ELSIF m_scopeArmIndex = m_matchedMasterArmIdx.right1ArmIdx OR m_scopeArmIndex = m_matchedMasterArmIdx.right2ArmIdx THEN
	// left arm
	// switch tele-controlled arm index when arm switch is triggerd
	IF m_armSwitch THEN
		IF m_teleSlaveArmIdx[1]=m_matchedMasterArmIdx.left1ArmIdx AND i_masterInputDataPool.m_slaveStatus.m_armState[m_matchedMasterArmIdx.left2ArmIdx]=SlaveArmState_InstruReady THEN
			nextTeleSlaveArmIdx[1] := m_matchedMasterArmIdx.left2ArmIdx;
		ELSIF 
			m_teleSlaveArmIdx[1]=m_matchedMasterArmIdx.left2ArmIdx AND i_masterInputDataPool.m_slaveStatus.m_armState[m_matchedMasterArmIdx.left1ArmIdx]=SlaveArmState_InstruReady THEN
			nextTeleSlaveArmIdx[1] := m_matchedMasterArmIdx.left1ArmIdx;
		ELSE
			IF  i_masterInputDataPool.m_slaveStatus.m_armState[m_matchedMasterArmIdx.left1ArmIdx]=SlaveArmState_InstruReady THEN
				nextTeleSlaveArmIdx[1] := m_matchedMasterArmIdx.left1ArmIdx;
			ELSIF i_masterInputDataPool.m_slaveStatus.m_armState[m_matchedMasterArmIdx.left2ArmIdx]=SlaveArmState_InstruReady THEN
				nextTeleSlaveArmIdx[1] := m_matchedMasterArmIdx.left2ArmIdx;
			ELSE
				nextTeleSlaveArmIdx[1] := m_matchedMasterArmIdx.left1ArmIdx;
			END_IF
		END_IF
	END_IF

	// right arm
	IF m_scopeArmIndex = m_matchedMasterArmIdx.right1ArmIdx THEN
		nextTeleSlaveArmIdx[2] := m_matchedMasterArmIdx.right2ArmIdx;
	ELSE
		nextTeleSlaveArmIdx[2] := m_matchedMasterArmIdx.right1ArmIdx;
	END_IF
END_IF

// check if arm-switch is triggerd
m_armSwitchFlag[1]:=m_teleSlaveArmIdx[1] <>  nextTeleSlaveArmIdx[1];
m_armSwitchFlag[2]:=m_teleSlaveArmIdx[2] <>  nextTeleSlaveArmIdx[2];

m_teleSlaveArmIdx:= nextTeleSlaveArmIdx;
END_METHOD

METHOD PROTECTED controllerTransit : BOOL
VAR_INPUT
END_VAR
VAR
	i :INT;
END_VAR
FOR i:=1 TO g_mArmNum DO 
	IF m_nextMasterArmState[i]<> m_masterArmState[i] THEN
		// reset current controller
		m_armCtrl[i].reset();
		
		// transit to new controller
		m_lastMasterArmState[i]:=m_masterArmState[i];
		m_masterArmState[i]:=m_nextMasterArmState[i];
		m_armCtrl[i]:=m_armCtrlFactory[i,m_masterArmState[i]];
		
		// init next controller
		m_armCtrl[i].Init(m_masterArms[i],m_armCtrlCmds[i]);
		
		// init scope controller
		IF m_masterArmState[i] = MasterArmState_Endoscope  THEN
			m_scopeCtrl.init(m_shoulderPoseInMonitor, m_masterArms, m_armCtrlCmds);
		END_IF
		
		m_masterArms[i].updateCmds(m_armCtrlCmds[i]);
	END_IF
END_FOR
END_METHOD

METHOD PUBLIC getStatus : BOOL
VAR_IN_OUT
	// master robot information, including arm status and cartesian data
	r_masterStatus :ST_MasterStatus;
	
	// master robot joint data
	r_masterJointsData :ST_MasterJointData;
	
END_VAR

VAR
	i:INT;
END_VAR
r_masterStatus.m_motionScale := m_motionScale;
r_masterStatus.m_armState:=m_masterArmState;
r_masterStatus.m_teleSlaveArmIdx := m_teleSlaveArmIdx;
r_masterStatus.m_matchedMasterArmIdx := m_matchedMasterArmIdx;

FOR i:=1 TO g_mArmNum DO
	// current info
	r_masterStatus.m_gripAngle[i]:=m_masterArms[i].gripAngle;
	// cartesion
	r_masterStatus.m_curArmPose[i]:=m_masterArms[i].curCartPose;
	r_masterStatus.m_curArmTwist[i]:=m_masterArms[i].curCartTwist;
	// joint
	r_masterJointsData.m_curMotorPos[i]:=m_masterArms[i].curMotorPos;
	r_masterJointsData.m_curLinkPos[i]:=m_masterArms[i].curLinkPos;
	r_masterJointsData.m_curJntPos[i]:=m_masterArms[i].curJntPos;
	r_masterJointsData.m_curJntVel[i]:=m_masterArms[i].curJntVel;
	r_masterJointsData.m_curJntTrq[i]:=m_masterArms[i].curJntTrq;
	r_masterJointsData.m_rawJntCurrent[i]:=m_masterArms[i].rawJntCurrent;
	r_masterJointsData.m_filtJntCurrent[i]:=m_masterArms[i].filtJntCurrent;
	
	// command info
	// cartesion
	r_masterStatus.m_cmdArmPose[i]:=m_masterArms[i].m_cmdCartPose;
	r_masterStatus.m_cmdArmTwist[i]:=m_masterArms[i].m_cmdCartTwist;
	// joint info
	r_masterJointsData.m_cmdJntPos[i]:=m_masterArms[i].m_cmdJntPos;
	r_masterJointsData.m_cmdJntVel[i]:=m_masterArms[i].m_cmdJntVel;
	r_masterJointsData.m_cmdJntTrq[i]:=m_masterArms[i].m_cmdJntTrq;
	r_masterJointsData.m_cmdJntCurrent[i]:=m_masterArms[i].cmdJntCurrent;
	//data to safety check
	r_masterStatus.m_gripHallSensor[i] := m_masterArms[i].m_gripHallSensorIO;
	r_masterStatus.m_slaveOnLine := m_slaveOnLine;
	r_masterStatus.m_IKSuccess[i] := m_armMatching[i].IKSuccess;
	r_masterStatus.m_timePeriod[i] := m_armMatching[i].timePeriod;
	//r_masterStatus.m_selfCheckStatus
END_FOR
END_METHOD

METHOD PUBLIC Init : BOOL
VAR_INPUT
END_VAR
VAR
	i:INT;
END_VAR
// init tele-controlled arm index
m_teleSlaveArmIdx[1]:=MatchedSlaveArmIdx_1;
m_teleSlaveArmIdx[2]:=MatchedSlaveArmIdx_3;

// shoulder pose in monitor
m_shoulderPoseInMonitor[1].m_pos[1]:=-g_shoulderDistance/2;
m_shoulderPoseInMonitor[2].m_pos[1]:=g_shoulderDistance/2;

FOR i:=1 TO g_mArmNum DO
	// arm init
	m_masterArms[i].Init(i);
	m_masterArmState[i]:=MasterArmState_Init;
	m_lastMasterArmState[i]:=MasterArmState_Init;
	m_nextMasterArmState[i]:=MasterArmState_Init;
	
	// command init
	m_armCtrlCmds[i].m_jntEnableFlag := g_zeroVec7i;
	m_armCtrlCmds[i].m_jntOPMode := g_allPosMode;
	m_armCtrlCmds[i].m_cmdCartPose := m_masterArms[i].curCartPose;
	m_armCtrlCmds[i].m_cmdCartTwist := g_zeroVec6d;
	m_armCtrlCmds[i].m_cmdJntPos := m_masterArms[i].curJntPos;
	m_armCtrlCmds[i].m_cmdJntVel := g_zeroVec7d;
	m_armCtrlCmds[i].m_cmdJntAcc := g_zeroVec7d;
	m_armCtrlCmds[i].m_cmdJntTrq := g_zeroVec7d;
	
	// generate controller factory
	m_armCtrlFactory[i,MasterArmState_Error] := m_armError[i];
	m_armCtrlFactory[i,MasterArmState_Init] := m_armInit[i];
	m_armCtrlFactory[i,MasterArmState_Home] := m_armHome[i];
	m_armCtrlFactory[i,MasterArmState_Standby] := m_armStandBy[i];
	m_armCtrlFactory[i,MasterArmState_Matching] := m_armMatching[i];
	m_armCtrlFactory[i,MasterArmState_Ready] := m_armReady[i];
	m_armCtrlFactory[i,MasterArmState_MasterSlave] := m_armMasterSlave[i];
	m_armCtrlFactory[i,MasterArmState_Clutch] := m_armClutch[i];
	m_armCtrlFactory[i,MasterArmState_Endoscope] := m_armEndoscope[i];
	m_armCtrlFactory[i,MasterArmState_Cart] := m_armCart[i];
	m_armCtrlFactory[i,MasterArmState_GravityCali] := m_armGravityCali[i];
	m_armCtrlFactory[i,MasterArmState_Test] := m_armTest[i];
	m_armCtrlFactory[i,MasterArmState_Disable] := m_armDisable[i];
	m_armCtrlFactory[i,MasterArmState_Performance] := m_armPerformance[i];

	// assign controller
	m_armCtrl[i]:=m_armCtrlFactory[i,m_masterArmState[i]];
	m_armCtrl[i].Init(m_masterArms[i],m_armCtrlCmds[i]);
	
	// init master-slave trigger
	m_MSCtrlTriggerCheck[i].init(g_armCtrlCycleTime, 2);
END_FOR
END_METHOD

METHOD PROTECTED MSCtrlTriggerCheck : BOOL
VAR_IN_OUT CONSTANT
		i_masterInputDataPool:ST_MasterInputDataPool;
END_VAR
VAR
	i:INT;
END_VAR
FOR i:=1 TO g_mArmNum DO
	IF MasterArmState_Ready = m_masterArmState[i] AND SlaveArmState_InstruReady = m_instruArmState[i] 
		AND SlaveArmState_ScopeReady = m_scopeArmState AND i_masterInputDataPool.m_cartStatus.m_surgonReady THEN
		m_MSCtrlTriggerFlag[i]:=m_MSCtrlTriggerCheck[i].run(m_masterArms[i].gripAngle);
	END_IF
	
	IF  MatchedSlaveArmIdx_NULL =  m_teleSlaveArmIdx[i] OR   NOT(i_masterInputDataPool.m_cartStatus.m_surgonReady) 
		OR 	NOT(i_masterInputDataPool.m_slaveStatus.m_instruStauts[m_teleSlaveArmIdx[i]].m_ready) 
		OR m_masterArmState[i] = MasterArmState_Error OR i_masterInputDataPool.m_cartStatus.m_consoleInAdjust
		OR  SlaveArmState_Error = m_instruArmState[i] OR SlaveArmState_Disable = m_instruArmState[i]  THEN
		m_MSCtrlTriggerFlag[i]:=FALSE;
		m_MSCtrlTriggerCheck[i].reset();
	END_IF  
END_FOR
END_METHOD

METHOD PUBLIC run : BOOL
VAR_IN_OUT CONSTANT
	i_masterInputDataPool:ST_MasterInputDataPool;
END_VAR
VAR
	i:INT;
END_VAR
m_motionScale := i_masterInputDataPool.m_UIData.m_motionScale;
m_monitorAngle := i_masterInputDataPool.m_cartStatus.m_monitorAngle;

// check slave connection
m_slaveOnLine := m_slaveOnLineCheck.check(i_masterInputDataPool.m_slaveStatus.m_slaveHeartBeat);

// update shoulder pose
updateShoulderPose();

// check tele-operated slave arms index
checkTeleSlaveArmIdx(i_masterInputDataPool);

// check if to trig ultrasonic knife ratotation clutch
USKnifeClutchCheck(i_masterInputDataPool);

// update arm status
FOR i:=1 TO g_mArmNum DO
	// update dynamic data
	m_masterArms[i].updateDyna(i_masterInputDataPool.m_masterDynaData);
								
	// update master arm kinematics
	m_masterArms[i].updateStatus();
END_FOR

// state machine transition
stateMachine(i_masterInputDataPool);

// controller transition
controllerTransit();

// run arm controller
FOR i:=1 TO g_mArmNum DO
	// null ptr check
	ASSERT(0 <> m_armCtrl[i]);
	
	// run controller
	m_armCtrl[i].run(m_teleSlaveArmIdx[i], m_shoulderPoseInMonitor[i], m_masterArms[i],
						i_masterInputDataPool.m_slaveStatus,m_armCtrlCmds[i]);
						
	// update commands to drivers
	m_masterArms[i].updateCmds(m_armCtrlCmds[i]);
END_FOR

// run scope controller
IF m_masterArmState[1] = MasterArmState_Endoscope AND m_masterArmState[2] = MasterArmState_Endoscope THEN
	m_scopeCtrl.run(m_teleSlaveArmIdx, m_shoulderPoseInMonitor, m_masterArms, i_masterInputDataPool.m_slaveStatus, m_armCtrlCmds);
	m_masterArms[1].updateCmds(m_armCtrlCmds[1]);
	m_masterArms[2].updateCmds(m_armCtrlCmds[2]);
END_IF
END_METHOD

PROPERTY shoulderPose : ARRAY[1..2] OF ST_Frame
GET
shoulderPose := m_shoulderPoseInMonitor;
END_GET
END_PROPERTY

// state machine check and transit 
METHOD PROTECTED stateMachine : BOOL
VAR_IN_OUT CONSTANT
		i_masterInputDataPool:ST_MasterInputDataPool;
END_VAR
VAR
	i:INT;
	enableClutch :BOOL;
END_VAR
// get instrument arm state
FOR i:=1 TO g_mArmNum DO
	IF MatchedSlaveArmIdx_NULL =  m_teleSlaveArmIdx[i] THEN
		m_instruArmState[i] := SlaveArmState_Error;
	ELSE
		m_instruArmState[i] := i_masterInputDataPool.m_slaveStatus.m_armState[m_teleSlaveArmIdx[i]];
	END_IF
END_FOR

// get endoscope arm state
m_scopeArmState := SlaveArmState_Error;
m_scopeArmIndex := MatchedSlaveArmIdx_null;
FOR i:=1 TO g_sArmNum DO 
	IF InstruType_endoscope =  i_masterInputDataPool.m_slaveStatus.m_instruStauts[i].m_type THEN
		m_scopeArmState := i_masterInputDataPool.m_slaveStatus.m_armState[i];
		m_scopeArmIndex := i;
		EXIT;
	END_IF
END_FOR

// check if master-slave grip angle match
MSCtrlTriggerCheck(i_masterInputDataPool);

// State machine transit 
FOR i:=1 TO g_mArmNum DO
	
	// flag if enable clutch
	enableClutch :=  i_masterInputDataPool.m_cartStatus.m_clutchSwitch OR (m_masterArms[i].handClutchSwitch AND i_masterInputDataPool.m_UIData.m_enableHandClutch);
	
	CASE m_masterArmState[i] OF
		// error
		MasterArmState_Error:
			// to standby
			IF FALSE = i_masterInputDataPool.m_safetyData.m_masterErrFlag[i] THEN
				IF m_armSelfCheckFinshedFlag[i] THEN
					m_nextMasterArmState[i] := MasterArmState_Standby;
				ELSE
					m_nextMasterArmState[i]:=MasterArmState_Home;
				END_IF
			END_IF
			
		// init
		MasterArmState_Init:
			// to home
			IF m_armCtrl[i].isFinished THEN
				// NOTICE: multiple cycles joints back to center during initialization
				// 			need to reset joints encoder data again
				m_masterArms[i].initJntPos();
				m_armSelfCheckFinshedFlag[i] := FALSE;
				m_nextMasterArmState[i]:=MasterArmState_Home;
			END_IF

		//home
		MasterArmState_Home:
			IF m_armCtrl[i].isFinished  THEN
				m_armSelfCheckFinshedFlag[i] := TRUE;
				m_nextMasterArmState[i]:=MasterArmState_Standby;
			END_IF
		
		//standby
		MasterArmState_Standby:
			// to matching
			IF SlaveArmState_InstruReady = m_instruArmState[i] AND SlaveArmState_ScopeReady = m_scopeArmState 
					AND i_masterInputDataPool.m_slaveStatus.m_asepticDeployCompleteFlag AND m_slaveOnLine THEN
				m_nextMasterArmState[i]:=MasterArmState_Matching;
			// to clutch
			ELSIF enableClutch THEN
				m_nextMasterArmState[i] := MasterArmState_Clutch; 
			// to cart
			ELSIF i_masterInputDataPool.m_cartStatus.m_monitorInAdjust THEN
				m_nextMasterArmState[i] := MasterArmState_Cart;
			END_IF
		
		//matching
		MasterArmState_Matching:
			// to ready
			IF m_armCtrl[i].isFinished THEN
				m_nextMasterArmState[i]:=MasterArmState_Ready;
			// to clutch
			ELSIF enableClutch THEN
				m_nextMasterArmState[i] := MasterArmState_Clutch; 
			// to standby
			ELSIF SlaveArmState_InstruReady <> m_instruArmState[i] OR SlaveArmState_ScopeReady <> m_scopeArmState
						OR m_armSwitchFlag[i] THEN
				m_nextMasterArmState[i]:=MasterArmState_Standby;
			// to cart
			ELSIF i_masterInputDataPool.m_cartStatus.m_monitorInAdjust THEN
				m_nextMasterArmState[i] := MasterArmState_Cart;
			END_IF
		
		//ready
		MasterArmState_Ready:
			// to standby
			IF SlaveArmState_InstruReady <> m_instruArmState[i] OR SlaveArmState_ScopeReady <> m_scopeArmState
					OR m_armSwitchFlag[i] THEN
				m_nextMasterArmState[i]:=MasterArmState_Standby;
			// to clutch
			ELSIF enableClutch THEN
				m_nextMasterArmState[i] := MasterArmState_Clutch; 
			// to cart
			ELSIF i_masterInputDataPool.m_cartStatus.m_monitorInAdjust THEN
				m_nextMasterArmState[i] := MasterArmState_Cart;
			// to master-slave
			ELSIF SlaveArmState_InstruReady = m_instruArmState[i] AND SlaveArmState_ScopeReady = m_scopeArmState 
					AND i_masterInputDataPool.m_cartStatus.m_surgonReady AND m_MSCtrlTriggerFlag[i] AND NOT(i_masterInputDataPool.m_cartStatus.m_consoleInAdjust) THEN
				m_nextMasterArmState[i] := MasterArmState_MasterSlave;
			ELSIF NOT i_masterInputDataPool.m_slaveStatus.m_asepticDeployCompleteFlag THEN
				m_nextMasterArmState[i]:=MasterArmState_Standby;
			END_IF
		
		//MasterSlave
		MasterArmState_MasterSlave:
			// to standdy
			IF  (SlaveArmState_InstruReady <> m_instruArmState[i] AND SlaveArmState_MasterSlave <> m_instruArmState[i])
				OR SlaveArmState_ScopeReady <> m_scopeArmState OR NOT(i_masterInputDataPool.m_cartStatus.m_surgonReady)
				OR m_armSwitchFlag[i] THEN
				m_nextMasterArmState[i]:=MasterArmState_Standby;
			// to clutch
			ELSIF enableClutch THEN
				m_nextMasterArmState[i] := MasterArmState_Clutch; 
			//to standby
			ELSIF NOT m_slaveOnLine THEN
				m_nextMasterArmState[i] := MasterArmState_Standby;
			END_IF
			
		//Clutch
		MasterArmState_Clutch:
			// to standby
			IF NOT(enableClutch) THEN
				m_nextMasterArmState[i]:=MasterArmState_Standby;
			END_IF
		
		// Endoscope 
		MasterArmState_Endoscope:
			// to standby
			IF NOT(i_masterInputDataPool.m_cartStatus.m_surgonReady) OR NOT(i_masterInputDataPool.m_cartStatus.m_endoscopeSwitch) 
				OR (SlaveArmState_ScopeReady <> m_scopeArmState AND SlaveArmState_EndoScope <> m_scopeArmState) THEN
				m_nextMasterArmState[i] := MasterArmState_Standby;
			// to clutch
			ELSIF enableClutch THEN
				m_nextMasterArmState[i] := MasterArmState_Clutch; 
			// to cart
			ELSIF i_masterInputDataPool.m_cartStatus.m_consoleInAdjust THEN
				m_nextMasterArmState[i] := MasterArmState_Cart;
			//to standby
			ELSIF NOT m_slaveOnLine THEN
				m_nextMasterArmState[i] := MasterArmState_Standby;
			END_IF
			
		// Cart 
		MasterArmState_Cart:
			// to standby
			IF NOT( i_masterInputDataPool.m_cartStatus.m_consoleInAdjust) THEN
				m_nextMasterArmState[i] := MasterArmState_Standby;
			END_IF
		
		//Gravity Calibration
		MasterArmState_GravityCali:
			// to standby
			IF  m_armCtrl[i].isFinished THEN
				m_nextMasterArmState[i]:=MasterArmState_Standby;
			END_IF
	
		//arm test
		MasterArmState_Test:
			// to standby
			IF  m_armCtrl[i].isFinished THEN
				m_nextMasterArmState[i]:=MasterArmState_Standby;
			END_IF
			
		//arm Performance
		MasterArmState_Performance:
			// to standby
			IF  m_armCtrl[i].isFinished THEN
				m_nextMasterArmState[i]:=MasterArmState_Standby;
			END_IF
			
		//arm disable
		MasterArmState_Disable:
			// to init
			IF  NOT(i_masterInputDataPool.m_UIData.m_masterArmDisableFlag[i]) THEN
				m_armSelfCheckFinshedFlag[i] := FALSE;
				m_nextMasterArmState[i]:=MasterArmState_Init;
			END_IF
	END_CASE
	
	// arm disable
	IF i_masterInputDataPool.m_UIData.m_masterArmDisableFlag[i] THEN
		m_nextMasterArmState[i] := MasterArmState_Disable;
	// error check
	ELSIF i_masterInputDataPool.m_safetyData.m_masterErrFlag[i] THEN
		m_nextMasterArmState[i] := MasterArmState_Error;
	END_IF
	
END_FOR

// To Endoscope Control 
IF SlaveArmState_ScopeReady = m_scopeArmState AND i_masterInputDataPool.m_cartStatus.m_endoscopeSwitch AND i_masterInputDataPool.m_cartStatus.m_surgonReady AND
  (MasterArmState_Standby = m_masterArmState[1] OR MasterArmState_Ready = m_masterArmState[1] OR MasterArmState_Matching = m_masterArmState[1] OR MasterArmState_MasterSlave = m_masterArmState[1]) AND 
  (MasterArmState_Standby = m_masterArmState[2] OR MasterArmState_Ready = m_masterArmState[2] OR MasterArmState_Matching = m_masterArmState[2] OR MasterArmState_MasterSlave = m_masterArmState[2]) THEN
	m_nextMasterArmState[1] := MasterArmState_Endoscope;
	m_nextMasterArmState[2] := MasterArmState_Endoscope;
END_IF
END_METHOD

METHOD PROTECTED updateShoulderPose : BOOL
VAR_INPUT
END_VAR
VAR
	monitorRot :mat3d;
END_VAR
// base monitor frame(0 rotation angle) in current monitor frame 
monitorRot := rotY( -m_monitorAngle);

// shoulder pose in current monitor frame
matMultiply(g_shoulderRotInMonitor,monitorRot, m_shoulderPoseInMonitor[1].m_rot);
m_shoulderPoseInMonitor[2].m_rot:=m_shoulderPoseInMonitor[1].m_rot;
END_METHOD

METHOD USKnifeClutchCheck : BOOL
VAR_IN_OUT CONSTANT
	i_masterInputDataPool:ST_MasterInputDataPool;
END_VAR

VAR
	i:INT;
END_VAR
FOR i:=1 TO g_sArmNum DO
	IF NOT(i_masterInputDataPool.m_slaveStatus.m_instruStauts[i].m_ready) THEN
		m_USKnifeRotClutch[i] := FALSE;
	END_IF
END_FOR

FOR i:=1 TO g_mArmNum DO
	IF (i_masterInputDataPool.m_slaveStatus.m_instruStauts[m_teleSlaveArmIdx[i]].m_type = InstruType_UltrasoundKnifeS OR i_masterInputDataPool.m_slaveStatus.m_instruStauts[m_teleSlaveArmIdx[i]].m_type = InstruType_UltrasoundKnifeU)
		AND  m_masterArmState[i] = MasterArmState_Clutch AND m_masterArms[i].handClutchSwitch THEN
		m_USKnifeRotClutch[m_teleSlaveArmIdx[i]] := TRUE;
	END_IF
END_FOR
END_METHOD

END_FUNCTION_BLOCK

// ---- SafetyCheck/Fb_SafetyCheck.TcPOU
FUNCTION_BLOCK Fb_SafetyCheck
VAR_INPUT
END_VAR
VAR_OUTPUT
END_VAR
VAR
	i, j:INT;
	m_checkDelay :ARRAY[1..g_maxNum] OF checkDelay;
	m_checkDelayTime :checkDelayTime;
	m_checkPermit:ARRAY[1..g_maxNum] OF  checkPermit;
	
	m_jntErrFlag:ARRAY[1..g_maxNum,0..g_maxArmJoint,1..3] OF BOOL;
	m_armErrFlag:ARRAY [1..g_maxNum,1..3] OF BOOL;
	m_errCode:UDINT;
	
	
	m_errNumType: ARRAY [1..3] OF INT;
	m_ArrayErrCodeType:ARRAY [1..3] OF ARRAY [0..100] OF UDINT;
	
	//The fault is sent to the UI at the frequency of 0.1S
	m_errCodeUpdateFlag: ARRAY [1..3] OF BOOL;
	m_errCodeUpdateTon: ARRAY [1..3] OF TON;
	
	m_curJntTorqueIOlast :ARRAY [1..g_maxArmNum] OF vec7di;  
	m_cmdJntPosLast : ARRAY [1..g_maxArmNum] OF vec7d;  
	m_cartCurJntTorqueIOlast :ARRAY [1..4] OF LREAL;  
	m_cartCmdJntPosLast : ARRAY [1..4] OF LREAL; 
	o_ErrCode:ARRAY [1..3] OF UDINT;
		
	//error robot data record
	m_dataRecord : Fb_dataRecord;
	
	m_PromptMassBusy:BOOL;
	m_PromptFlag:ARRAY[1..g_maxNum,1..20] OF UINT;
	m_deleteCode:UDINT;
	
END_VAR


VAR CONSTANT
	m_codeUpdateDelay:TIME:=T#0.1S;
	
	//Fault level: 1 indicates  prompt message, 2 indicates a recoverable fault and 3 indicates an unrecoverable fault
	m_promptMessageLevel : UINT :=1;
	m_rcvLevel : UINT :=2;
	m_unrcvLevel : UINT :=3;
END_VAR

METHOD armSafetyCheck : BOOL
VAR_INPUT
	i_armId:UDINT;
	i_safetyCheckVar :ARRAY[1..g_maxNum] OF checkInputVariable;
	i_masterStatus :ST_MasterStatus;
	i_masterJointData : ST_MasterJointData;
END_VAR

VAR
	k:INT;
END_VAR

//驱动器状态监测、驱动器未连接
FOR i:=1 TO g_mJntNum BY 1 DO
	m_checkDelay[i_ArmId].T_jntStatusErr[i](IN:= (i_safetyCheckVar[i_ArmId].m_masterDriverInput[i].m_statusWord=0 AND m_checkPermit[i_ArmId].m_jntStatusErr[i]), PT:=m_checkDelayTime.Ti_jntStatusErr , Q=> , ET=> );
	IF m_checkDelay[i_ArmId].T_jntStatusErr[i].Q  THEN
		errCodeAssign(i_ArmId, i_ArmId,  0, i, 16#3002 ,m_unrcvLevel );
	END_IF
END_FOR



//关节编码器监测
FOR i:=1 TO g_mJntNum BY 1 DO
	m_checkDelay[i_ArmId].T_linkEncErr[i](IN:= (i_safetyCheckVar[i_ArmId].m_masterDriverInput[i].m_linkEncoder=g_maxLinkEnc OR i_safetyCheckVar[i_ArmId].m_masterDriverInput[i].m_linkEncoder=g_minLinkEnc) AND m_checkPermit[i_ArmId].m_linkEncErr[i], PT:=m_checkDelayTime.Ti_linkEncErr , Q=> , ET=> );
	IF m_checkDelay[i_ArmId].T_linkEncErr[i].Q THEN
		errCodeAssign(i_ArmId, i_ArmId,  0, i,  16#3003 ,m_unrcvLevel );
	END_IF
END_FOR


//驱动器错误检测
FOR i:=1 TO g_mJntNum BY 1 DO
	m_checkDelay[i_ArmId].T_DriveErr[i](IN:= (i_safetyCheckVar[i_ArmId].m_masterDriverInput[i].m_driverError AND 16#20)=g_driveErrWord AND m_checkPermit[i_ArmId].m_driveErr[i] , PT:=m_checkDelayTime.Ti_driveErr , Q=> , ET=> );
	IF m_checkDelay[i_ArmId].T_DriveErr[i].Q THEN
		errCodeAssign(i_ArmId, i_ArmId,  0, i, 16#3004 ,m_unrcvLevel );
	END_IF
END_FOR


//双编码器偏差过大检测
FOR i:=1 TO g_mJntNum BY 1 DO
	m_checkDelay[i_ArmId].T_armJntEncErr[i](IN:= ABS(i_masterJointData.m_curLinkPos[i_armId][i]-i_masterJointData.m_curJntPos[i_armId][i])>=g_armMaxJntEncErr[i] AND m_checkPermit[i_ArmId].m_armJntEncErr[i], PT:=m_checkDelayTime.Ti_armJntEncErr , Q=> , ET=> );
	IF m_checkDelay[i_ArmId].T_armJntEncErr[i].Q THEN
		errCodeAssign( i_ArmId, i_ArmId,  0, i, 16#3005, m_unrcvLevel );
	END_IF
END_FOR


//关节运动超限位
FOR i:=1 TO g_mJntNum BY 1 DO
	m_checkDelay[i_armId].T_outOfLimit[i](IN:= i_masterJointData.m_curJntPos[i_armId][i]>= (g_maxJntPos[i_armId,i] + g_armJntPosLimitBuffer[i]) OR i_masterJointData.m_curJntPos[i_armId][i]<=(g_minJntPos[i_armId,i] - g_armJntPosLimitBuffer[i]) AND m_checkPermit[i_ArmId].m_outOfLimit[i], PT:=m_checkDelayTime.Ti_outofLimit , Q=> , ET=> );
	IF m_checkDelay[i_armId].T_outOfLimit[i].Q THEN
		errCodeAssign(i_armId, i_ArmId,  0, i, 16#3006, m_unrcvLevel );
	END_IF
END_FOR


//驱动器内部通讯错误
FOR i:=1 TO g_mJntNum BY 1 DO
	m_checkDelay[i_armId].T_currentIsNotUpdate[i](IN:= (i_safetyCheckVar[i_ArmId].m_masterDriverInput[i].m_current=m_curJntTorqueIOlast[i_ArmId][i] AND m_checkPermit[i_ArmId].m_currentIsNotUpdate[i]), PT:=m_checkDelayTime.Ti_currentIsNotUpdate , Q=> , ET=> );
	IF  m_checkDelay[i_armId].T_currentIsNotUpdate[i].Q THEN
		errCodeAssign(i_armId, i_ArmId,  0, i, 16#3009 ,m_unrcvLevel );
	END_IF
	m_curJntTorqueIOlast[i_armId][i]:=i_safetyCheckVar[i_armId].m_masterDriverInput[i].m_current;
END_FOR


//关节跟随误差过大
//FOR i:=1 TO g_mJntNum BY 1 DO
//	m_checkDelay[i_ArmId].T_armJntFollowErr[i](IN:= ABS(i_masterJointData.m_cmdJntPos[i_armId][i]- i_masterJointData.m_curJntPos[i_armId][i])>g_armMaxJntFollowErr[i]  AND m_checkPermit[i_ArmId].m_armJntFollowErr[i], PT:=m_checkDelayTime.Ti_armJntFollowErr , Q=> , ET=> );
//	IF m_checkDelay[i_ArmId].T_armJntFollowErr[i].Q THEN
//		errCodeAssign(i_ArmId, i_ArmId,  0, i, 16#2002, m_rcvLevel );
//	END_IF
//END_FOR


//笛卡尔空间指令与位置偏差检测
//FOR i:=1 TO 6 BY 1 DO
//	m_checkDelay[i_ArmId].T_spacePoseErr[i](IN:= i_safetyCheckVar[i_ArmId].m_spacePoseErr[i]> g_maxCartPoseErr[i] AND m_checkPermit[i_ArmId].m_spacePoseErr[i], PT:=m_checkDelayTime.Ti_spacePoseErr , Q=> , ET=> );
//	IF m_checkDelay[i_ArmId].T_spacePoseErr[i].Q THEN
//		errCodeAssign(i_ArmId, i_ArmId, 1, i, 16#2004, m_rcvLevel );
//	END_IF
//END_FOR


//current overrun check
FOR i:=1 TO g_mJntNum BY 1 DO
	m_checkDelay[i_armId].T_jntCurrentErr[i](IN:= ABS(i_safetyCheckVar[i_armId].m_motorCurrentIntegral[i])>g_motorCurrentLimit[i] AND m_checkPermit[i_ArmId].m_jntCurrentErr[i], PT:=m_checkDelayTime.Ti_jntCurrentErr , Q=> , ET=> );
	IF m_checkDelay[i_armId].T_jntCurrentErr[i].Q THEN
		errCodeAssign(i_armId, i_ArmId,  0, i, 16#2005, m_rcvLevel );
	END_IF
END_FOR


//Ethercat communication check
FOR i:=1 TO g_mJntNum BY 1 DO
	IF NOT i_safetyCheckVar[i_ArmId].m_EtherCATState[i].EtherCATState THEN
		errCodeAssign(i_ArmId, i_ArmId, 0, i, 16#2006, m_rcvLevel );
	END_IF
END_FOR


//self check failure
IF i_masterStatus.m_armState[i_armId] = MasterArmState_Home AND i_masterStatus.m_timePeriod[i] > g_selfCheckTimeLimit THEN//i_safetyCheckVar[i_armId].m_selfCheckFail THEN
	errCodeAssign(i_armId, i_ArmId,  0, 0, 16#2010, m_rcvLevel );
END_IF

//motor encoder mutation detection
FOR i:=1 TO g_mJntNum BY 1 DO
	IF i_safetyCheckVar[i_armId].m_motorEncSaltaValue[i]>g_maxJntCurSalta[i] THEN
		errCodeAssign(i_armId, i_ArmId, 0, i, 16#200C, m_rcvLevel );
	END_IF
END_FOR

//master hall anomaly
IF i_masterStatus.m_gripHallSensor[i_armId] = 0 THEN
	errCodeAssign(i_armId, i_ArmId, 0, 0, 16#200E, m_rcvLevel );
END_IF
END_METHOD

METHOD arrayDeleteFrist : ARRAY [0..100] OF UDINT;
VAR_INPUT
	i_array:ARRAY [0..100] OF UDINT;
END_VAR

VAR
	k:INT;
END_VAR

arrayDeleteFrist[100]:=0;

FOR k:=0 TO 99 BY 1 DO
	arrayDeleteFrist[k]:=i_array[k+1];
END_FOR
END_METHOD

METHOD arrayDeleteInput : BOOL
VAR_INPUT
	i_Array:ARRAY[0..100] OF UDINT;
	i_DeleteCode:UDINT;
END_VAR

VAR_OUTPUT
	o_Array:ARRAY[0..100] OF UDINT;
	
END_VAR

VAR
	i:INT;
	Falg:BOOL;
END_VAR

FOR i:=0 TO 20 BY 1 DO 
	IF i_Array[i]=i_DeleteCode THEN
		Falg:=TRUE;
	END_IF
	
	IF Falg=TRUE THEN
		o_Array[i]:=i_Array[i+1];
	ELSE
		o_Array[i]:=i_Array[i];
	END_IF
END_FOR
o_Array[20]:=0;
END_METHOD

METHOD arrayFIFO : ARRAY [0..100] OF  UDINT
VAR_INPUT
	i_array:ARRAY[0..100] OF UDINT;
	i_newData:UDINT;
END_VAR

VAR
	i:INT;
END_VAR

FOR i:=0 TO 20 BY 1 DO
	arrayFIFO[i+1]:=i_array[i];
END_FOR

arrayFIFO[0]:=i_newData;
END_METHOD

METHOD arrayFILO : ARRAY [0..100] OF  UDINT
VAR_INPUT
	i_array:ARRAY[0..100] OF UDINT;
	i_newData:UDINT;
END_VAR

VAR
	i:INT;
END_VAR

FOR i:=0 TO 99 BY 1 DO
	arrayFILO[i]:=i_array[i];
	IF i_array[i]=0 THEN
		arrayFILO[i]:=i_newData;
		EXIT;
	END_IF
END_FOR
END_METHOD

METHOD cartSafetyCheck : BOOL
VAR_INPUT
	i_armId:UDINT;
	i_safetyCheckVar : checkInputVariable;
	i_cartJointData : ST_CartJointData;
END_VAR


VAR
	k:INT;
END_VAR


//驱动器状态监测、驱动器未连接
FOR i:=1 TO g_maxCartJoint BY 1 DO
	m_checkDelay[i_armId].T_cartJntStatusErr[i](IN:= (i_safetyCheckVar.m_cartDriverInput[i].m_statusWord=0 AND m_checkPermit[i_ArmId].m_cartJntStatus[i]), PT:=m_checkDelayTime.Ti_CarJntStatus , Q=> , ET=> );
	IF m_checkDelay[i_armId].T_cartJntStatusErr[i].Q THEN
		errCodeAssign(i_armId, i_ArmId,  0, i, 16#3002 ,m_unrcvLevel );
	END_IF
END_FOR



//关节编码器监测
FOR i:=1 TO g_maxCartJoint BY 1 DO
	m_checkDelay[i_armId].T_cartLinkEncErr[i](IN:= (i_safetyCheckVar.m_cartDriverInput[i].m_linkEncoder=g_cartMaxLinkEnc[i] OR i_safetyCheckVar.m_cartDriverInput[i].m_linkEncoder=g_cartMinLinkEnc[i]) AND m_checkPermit[i_ArmId].m_cartJntEncErr[i], PT:=m_checkDelayTime.Ti_CarActSec , Q=> , ET=> );
	IF m_checkDelay[i_armId].T_cartLinkEncErr[i].Q THEN
		errCodeAssign(i_armId, i_ArmId,  0, i, 16#3003 ,m_unrcvLevel );
	END_IF
END_FOR


//驱动器错误检测
FOR i:=1 TO g_maxCartJoint BY 1 DO
	m_checkDelay[i_armId].T_cartDriveErr[i](IN:= (i_safetyCheckVar.m_cartDriverInput[i].m_driverError AND 16#20)=32 AND m_checkPermit[i_ArmId].m_cartDriveErr[i] , PT:=m_checkDelayTime.Ti_CarDriveErr , Q=> , ET=> );
	IF m_checkDelay[i_armId].T_cartDriveErr[i].Q THEN
		errCodeAssign(i_armId, i_ArmId,  0, i, 16#3004 ,m_unrcvLevel );
	END_IF
END_FOR



//台车双编码器偏差过大
FOR i:=1 TO g_maxCartJoint BY 1 DO
	m_checkDelay[i_armId].T_cartJntEncErr[i](IN:= ABS (i_cartJointData.m_curLinkPos[i]-i_cartJointData.m_curJntPos[i])>g_cartMaxJntEncErr[i] AND m_checkPermit[i_ArmId].m_cartJntEncErr[i], PT:=m_checkDelayTime.Ti_CarDualEncDev , Q=> , ET=> );
	IF m_checkDelay[i_armId].T_cartJntEncErr[i].Q THEN
		errCodeAssign(i_armId, i_ArmId,  0, i, 16#3005 ,m_unrcvLevel );
	END_IF
END_FOR


//关节运动超限位
FOR i:=1 TO g_maxCartJoint BY 1 DO
	m_checkDelay[i_armId].T_cartOutOfLimit[i](IN:= (i_cartJointData.m_curJntPos[i]>=g_cartMaxJntLimit[i] OR i_cartJointData.m_curJntPos[i]<=g_cartMinJntLimit[i]) AND m_checkPermit[i_ArmId].m_cartOutOfLimit[i] , PT:=m_checkDelayTime.Ti_CaroutofLimit , Q=> , ET=> );
	IF m_checkDelay[i_armId].T_cartOutOfLimit[i].Q THEN
		errCodeAssign(i_armId, i_ArmId,  0, i, 16#3006 ,m_unrcvLevel );
	END_IF
END_FOR


//驱动器内部通讯错误
FOR i:=1 TO g_maxCartJoint BY 1 DO
	m_checkDelay[i_armId].T_cartCurrentIsNotUpdate[i](IN:= (i_safetyCheckVar.m_cartDriverInput[i].m_current=m_cartCurJntTorqueIOlast[i] AND m_checkPermit[i_ArmId].m_cartCurrentIsNotUpdate[i]), PT:=m_checkDelayTime.Ti_CarTorMotor , Q=> , ET=> );
	IF m_checkDelay[i_armId].T_cartCurrentIsNotUpdate[i].Q THEN
		errCodeAssign(i_armId, i_ArmId,  0, i, 16#3009 ,m_unrcvLevel );
	END_IF
	m_cartCurJntTorqueIOlast[i]:=i_safetyCheckVar.m_cartDriverInput[i].m_current;
END_FOR


//关节跟随误差过大
FOR i:=1 TO g_maxCartJoint BY 1 DO
	m_checkDelay[i_armId].T_cartJntFollowErr[i](IN:= ABS(i_cartJointData.m_cmdJntPos[i]- i_cartJointData.m_curJntPos[i])>g_cartMaxJntFollowErr[i]  AND m_checkPermit[i_ArmId].m_cartFollowErr[i], PT:=m_checkDelayTime.Ti_CarFollowDev , Q=> , ET=> );
	IF m_checkDelay[i_armId].T_cartJntFollowErr[i].Q THEN
		errCodeAssign(i_armId, i_ArmId,  0, i, 16#2002 ,m_rcvLevel );
	END_IF
END_FOR


//关节速度监控
FOR i:=1 TO g_maxCartJoint BY 1 DO
	m_checkDelay[i_armId].T_cartJntVelErr[i](IN:= ABS(i_cartJointData.m_curJntVel[i])>g_cartMaxJntVel[i] AND m_checkPermit[i_ArmId].m_cartJntVelErr[i], PT:=m_checkDelayTime.Ti_CarJntVel , Q=> , ET=> );
	IF m_checkDelay[i_armId].T_cartJntVelErr[i].Q THEN
		errCodeAssign(i_armId, i_ArmId,  0, i, 16#2003 ,m_rcvLevel );
	END_IF
END_FOR


//电流超限监测
FOR i:=1 TO g_maxCartJoint BY 1 DO
	m_checkDelay[i_armId].T_cartJntCurrentErr[i](IN:= ABS(i_cartJointData.m_curJntTrq[i])>g_cartMaxJntCurrent[i] AND m_checkPermit[i_ArmId].m_cartJntCurrentErr[i], PT:=m_checkDelayTime.Ti_CarJntCurrent , Q=> , ET=> );
	IF m_checkDelay[i_armId].T_cartJntCurrentErr[i].Q THEN
		errCodeAssign(i_armId, i_ArmId,  0, i, 16#2005 ,m_rcvLevel );
	END_IF
END_FOR


//Ethercat通讯检测
FOR i:=1 TO g_maxCartJoint BY 1 DO
	IF NOT i_safetyCheckVar.m_cartEtherCATState[i].EtherCATState THEN
		errCodeAssign(i_armId, i_ArmId,  0, i, 16#2006 ,m_rcvLevel );
	END_IF
END_FOR
END_METHOD

PROPERTY checkPermit : REFERENCE TO ARRAY[1..g_maxNum] OF  checkPermit
GET
checkPermit ref= m_checkPermit;
END_GET
SET
END_SET
END_PROPERTY

METHOD electriAngleDev : DINT
VAR_INPUT
	i_motorElectriAngleDev : DINT;
END_VAR

IF i_motorElectriAngleDev > 50000 THEN
	electriAngleDev := i_motorElectriAngleDev - 65535;
ELSIF i_motorElectriAngleDev < -50000 THEN
	electriAngleDev := i_motorElectriAngleDev + 65535;
ELSE
	electriAngleDev := i_motorElectriAngleDev;
END_IF
END_METHOD

METHOD errCodeAssign : BOOL
VAR_INPUT
	i_armId:UDINT;
	i_errLocation:UDINT;
	i_errCodeMode:UDINT;
	i_errJoint:UDINT;
	i_errID:UDINT;
	i_errFlagID :UINT;
END_VAR
IF m_jntErrFlag[i_armId,i_errJoint,i_errFlagID]=FALSE THEN
	m_jntErrFlag[i_armId,i_errJoint,i_errFlagID]:=TRUE;
	m_errCode:=SHL(i_errLocation,24)+SHL(i_errCodeMode,20)+SHL(i_errJoint,16)+i_errID;
	
	
	IF i_errID>=16#3000 THEN
		m_errNumType[m_unrcvLevel]:=LIMIT(0,m_errNumType[m_unrcvLevel]+1,100);
		m_arrayErrCodeType[m_unrcvLevel][m_errNumType[m_unrcvLevel]]:=m_errCode;
		g_arrayErrCodeArm[i_armId]:=arrayFILO(i_Array:= g_arrayErrCodeArm[i_ArmId], i_NewData:=m_errCode );
		m_armErrFlag[i_armId,m_unrcvLevel]:=TRUE;
		
	ELSIF i_errID>=16#2000 THEN
		m_errNumType[m_rcvLevel]:=LIMIT(0,m_errNumType[m_rcvLevel]+1,100);
		m_arrayErrCodeType[m_rcvLevel][m_errNumType[m_rcvLevel]]:=m_errCode;
		g_arrayErrCodeArm[i_armId]:=arrayFILO(i_Array:= g_arrayErrCodeArm[i_ArmId], i_NewData:=m_errCode );
		m_armErrFlag[i_armId,m_rcvLevel]:=TRUE;
		
	END_IF
END_IF
END_METHOD

METHOD errCodeUpdating :ARRAY [1..3] OF UDINT;
VAR_INPUT
END_VAR

m_errCodeUpdateTon[m_unrcvLevel](IN:= NOT m_errCodeUpdateFlag[3], PT:=m_codeUpdateDelay , Q=> m_errCodeUpdateFlag[3], ET=> );
IF m_errCodeUpdateFlag[m_unrcvLevel] THEN
	IF m_errNumType[m_unrcvLevel]>=1 THEN
		m_ArrayErrCodeType[m_unrcvLevel]:=ArrayDeleteFrist(i_Array:=m_ArrayErrCodeType[3]) ;
		o_ErrCode[m_unrcvLevel]:=m_ArrayErrCodeType[m_unrcvLevel][0] ;
		g_ArrayErrCodeTypeTest[m_unrcvLevel]:=arrayFILO(i_Array:= g_ArrayErrCodeTypeTest[m_unrcvLevel], i_NewData:=o_ErrCode[m_unrcvLevel] );
		m_errNumType[m_unrcvLevel]:=m_errNumType[m_unrcvLevel]-1;
	END_IF
END_IF


m_errCodeUpdateTon[m_rcvLevel](IN:= NOT m_errCodeUpdateFlag[2], PT:=m_codeUpdateDelay , Q=> m_errCodeUpdateFlag[2], ET=> );
IF m_errCodeUpdateFlag[m_rcvLevel] THEN
	IF m_errNumType[m_rcvLevel]>=1 THEN
		m_ArrayErrCodeType[m_rcvLevel]:=ArrayDeleteFrist(i_Array:=m_ArrayErrCodeType[m_rcvLevel]) ;
		o_ErrCode[m_rcvLevel]:=m_ArrayErrCodeType[m_rcvLevel][0] ;
		g_ArrayErrCodeTypeTest[m_rcvLevel]:=arrayFILO(i_Array:= g_ArrayErrCodeTypeTest[m_rcvLevel], i_NewData:=o_ErrCode[m_rcvLevel] );
		m_errNumType[m_rcvLevel]:=m_errNumType[m_rcvLevel]-1;
	END_IF
END_IF
END_METHOD

METHOD errFlagReset : BOOL
VAR_INPUT
END_VAR

FOR i := 1 TO g_maxNum DO
	FOR j :=0 TO g_maxArmJoint DO
		m_jntErrFlag[i, j, 2]:=FALSE;
	END_FOR
	m_armErrFlag[i, 2]:=FALSE;
END_FOR

o_ErrCode[2]:=0;
END_METHOD

METHOD poseErrCheck : vec6d
VAR_INPUT
	i_cmdPose : ST_Frame;
	i_curPose :ST_Frame;
END_VAR

VAR
	posErr,oriErr:Vec3d;
	matT,rotErr:Mat3d;
	errAngle :LREAL;
	errAxis :Vec3d;
	i : INT;
END_VAR
vecSub(i_cmdPose.m_pos, i_curPose.m_pos,posErr);

matTranspose(i_cmdPose.m_rot, matT);
matMultiply(matT,i_curPose.m_rot, rotErr);
rot2AngAxis(rotErr, angle=>errAngle, axis=>errAxis);
vecMultiNum(errAxis, errAngle,oriErr);

FOR i := 1 TO 6 DO
	IF i <= 3 THEN
		poseErrCheck[i] := posErr[i];
	ELSE
		poseErrCheck[i] := oriErr[i];
	END_IF
END_FOR
END_METHOD

METHOD promptMassCode : BOOL
VAR_INPUT
	i_PromptStatus:BOOL;
	i_ArmId:UDINT;
	i_ErrID:UDINT;
	i_ErrLocation:UDINT;
END_VAR

m_PromptMassBusy:=TRUE;

//提示置位
IF i_PromptStatus=TRUE AND m_PromptFlag[i_ArmId,i_ErrID]=0 THEN
	m_PromptFlag[i_ArmId,i_ErrID]:=1;
END_IF

//输出提示故障码
IF m_PromptFlag[i_ArmId,i_ErrID]=1 THEN
	m_ErrCode:=SHL(i_ErrLocation,24)+i_ErrID+16#1010;
	m_ArrayErrCodeType[1]:=ArrayFIFO(i_Array:= m_ArrayErrCodeType[1], i_NewData:=m_ErrCode );//m_ErrCode;
	m_PromptFlag[i_ArmId,i_ErrID]:=2;
END_IF

//清除提示故障码
IF m_PromptFlag[i_ArmId,i_ErrID]=2 AND i_PromptStatus=FALSE THEN
	m_deleteCode:=SHL(i_ErrLocation,24)+i_ErrID+16#1010;
	ArrayDeleteInput(i_Array:= m_ArrayErrCodeType[1], i_DeleteCode:=m_deleteCode , o_Array=> m_ArrayErrCodeType[1]);
	m_PromptFlag[i_ArmId,i_ErrID]:=0;
END_IF
o_ErrCode[1]:=m_ArrayErrCodeType[1][0];
m_PromptMassBusy:=FALSE;
END_METHOD

METHOD systemSafetyCheck : BOOL
VAR_INPUT
	i_armId:UDINT;
	i_safetyCheckVar :ARRAY[1..g_maxNum] OF checkInputVariable;
	i_masterStatus :ST_MasterStatus;
	i_cartJointData : ST_CartJointData;
	i_masterJointData : ST_MasterJointData;
END_VAR

VAR
	k:INT;
END_VAR
IF i_armId =g_cartNum THEN 
	//cart safrty check
	cartSafetyCheck(i_armId,i_safetyCheckVar[i_armId],i_cartJointData);
ELSE
	//master arms safety check
	armSafetyCheck(i_armId,i_safetyCheckVar,i_masterStatus,i_masterJointData);
END_IF

//StopButton
IF  i_safetyCheckVar[i_ArmId].PCStopButton=0 OR NOT i_safetyCheckVar[i_ArmId].MasterStopButton OR i_safetyCheckVar[i_ArmId].SlaveStopButton THEN
	errCodeAssign(i_ArmId, 16#0B, 0, 0, 16#2001, m_rcvLevel );
END_IF

//prompt message
FOR i:=1 TO 10 DO
	PromptMassCode( i_safetyCheckVar[i_ArmId].m_promptStatus[i], i_ArmId,  i,  i_safetyCheckVar[i_ArmId].m_promptLocation[i]);
END_FOR
END_METHOD

END_FUNCTION_BLOCK
